{warning 'TODO: Remove all instances of bBusy and remove from VAR list in FB_StateMachine'}
FUNCTION_BLOCK FB_StateMachine IMPLEMENTS I_StateMachine
VAR_INPUT
	bActive : BOOL := TRUE;
	bErrorAck : BOOL;
	eStateSourceID : E_StateSourceID;
	
	aErrorLog : REFERENCE TO ARRAY[1..SystemConfig.MAIN_EVENT_LOG_MAX_LENGTH] OF ST_Event; //Reference to the event array initially created in MAIN
	nErrorLogIndex : REFERENCE TO UINT; //Reference to the logging index initially defined in MAIN, should be 0 at the beginning of each PLC cycle
END_VAR

VAR
	// Outer-Case State Tracking Variables
	eOuterLoopState : E_OuterLoopSM_States;
	sOuterLoopState : T_MaxString := '';
	nLastOuterLoopState : UINT := 0;	
	nOuterTempState : UINT := 0;
	sLastOuterLoopState : T_MaxString := '';
	
	// Inner-Case State Tracking Variables
	nInnerLoopState : REFERENCE TO UINT;
	sInnerLoopState : T_MaxString := '';
	nLastInnerLoopState : UINT := 0;
	nInnerTempState : UINT := 0;
	sLastInnerLoopState : T_MaxString := '';
	
	// DB Logging Stuff
	eStateMachineSourceID : E_StateSourceID;
	fbEventHandler : FB_EventHandler;
	sEventTrace	: T_MaxString := '';
	
	bBusy : BOOL;
	
//	bEnableOuterStateChanges : BOOL := SystemConfig.ENABLE_OUTER_STATE_CHANGES;
//	bEnableInnerStateChanges : BOOL := SystemConfig.ENABLE_INNER_STATE_CHANGES;
END_VAR

VAR_OUTPUT
	bError : BOOL;
	sErrorDetails : T_MaxString;			
	nErrorInTask : UINT;			
END_VAR

PROPERTY Active : BOOL
GET
Active := THIS^.bActive;
END_GET
SET
bActive := Active;
END_SET
END_PROPERTY

PROPERTY PUBLIC Busy : BOOL
GET
//Busy := isBusy();

(*
	Returns THIS^.bBusy in all cases except:
	1. We are enabled/active and transitioning to Operational - This will return FALSE until operational
	2. We are enabled/active and in Setup.
	3. We are enabled/active and in either DisablingError or DisablingInactive
*)

IF bActive THEN
	
	IF eOuterLoopState = E_OuterLoopSM_States.DisabledError THEN
		Busy := FALSE; // Not busy when active and waiting for error ack 
	ELSIF eOuterLoopState <> E_OuterLoopSM_States.Operational THEN
		Busy := TRUE; // Busy if we are active and not operational
	ELSE 
		Busy := (nInnerLoopState <> 0); // Busy In operational, if we are not idle
	END_IF
	
ELSE // NOT bActive
	
	IF eOuterLoopState = E_OuterLoopSM_States.Inactive THEN
		IF nOuterTempState =  E_OuterLoopSM_States.Inactive THEN
			Busy := FALSE; // Busy until we spend at least 1 cycle inactive
		ELSE
			Busy := TRUE; // We have spent at least 1 cycle inactive
		END_IF
	ELSIF eOuterLoopState = E_OuterLoopSM_States.DisabledError THEN
		Busy := FALSE; // Not busy while waiting for error ack
	ELSE
		Busy := TRUE; // Busy until we reach inactive state
	END_IF
	
END_IF
END_GET
END_PROPERTY

METHOD ChangeInnerState : BOOL
VAR_INPUT
	nNewState : UINT;
END_VAR
nInnerLoopState := nNewState;
END_METHOD

METHOD ChangeOuterState : BOOL
VAR_INPUT
	nNewState	: E_OuterLoopSM_States;
END_VAR
eOuterLoopState := nNewState;
END_METHOD

(*
Use the method as Case Variable ->
CASE CyclicInnerCase(TO_String(enum)) OF
1: ;
2: ;
ELSE ;
END_CASE
*)
METHOD PROTECTED CyclicInnerCase : UINT
VAR_INPUT
    sState : T_MaxString;//Name of the current state (TO_String(enum))
END_VAR
VAR_INST
    bInit : BOOL := TRUE;
END_VAR


IF (THIS^.nInnerTempState <> THIS^.nInnerLoopState) OR bInit THEN	
	// Save PreviousState
	IF bInit THEN
//		THIS^.nInnerLoopState := 0;
		THIS^.nLastInnerLoopState := THIS^.nInnerLoopState;
		THIS^.sLastInnerLoopState := sState;
		bInit := FALSE;
	ELSE
		THIS^.nLastInnerLoopState := THIS^.nInnerTempState;
		THIS^.sLastInnerLoopState := THIS^.sInnerLoopState;
		bInit := FALSE;
	END_IF
	
	// Save active State
	nInnerTempState := nInnerLoopState; 
	THIS^.sInnerLoopState := sState; //save aktive state string
	IF SystemConfig.ENABLE_INNER_STATE_CHANGES THEN
		fbEventHandler.SaveState(sLastState:=sLastInnerLoopState, sNewState:=sState, bOuter:=FALSE); //Logging after the new state has been adopted
	END_IF
END_IF


CyclicInnerCase := nInnerLoopState; //return state
END_METHOD

(*
Use the method as Case Variable ->
CASE CyclicOuterCase(TO_String(enum)) OF
1: ;
2: ;
ELSE ;
END_CASE
*)

{attribute 'monitoring':='variable'}
METHOD PRIVATE CyclicOuterCase : UINT
VAR_INPUT
    sState : T_MaxString;//Name of the current state (TO_String(enum))
END_VAR
VAR_INST
    bInit : BOOL := TRUE;
END_VAR
	
IF (THIS^.nOuterTempState <> THIS^.eOuterLoopState) OR bInit THEN

	// Save PreviousState
	IF bInit THEN
		THIS^.nLastOuterLoopState := THIS^.eOuterLoopState;
		THIS^.sLastOuterLoopState := sState;
	ELSE
		THIS^.nLastOuterLoopState := THIS^.nOuterTempState;
		THIS^.sLastOuterLoopState := THIS^.sOuterLoopState;
	END_IF
	// Save active State
	nOuterTempState := eOuterLoopState; 
	THIS^.sOuterLoopState := sState; //save aktive state string
	IF bInit THEN
		// Skips first outer state transition into setup.
		bInit := FALSE;
		
	ELSIF SystemConfig.ENABLE_OUTER_STATE_CHANGES THEN 
		fbEventHandler.SaveState(sLastState:=sLastOuterLoopState, sNewState:=sState, bOuter:=TRUE); //Logging after the new state has been adopted
	END_IF
	
END_IF


CyclicOuterCase := eOuterLoopState; //return state
END_METHOD

METHOD Disable : BOOL
// Default SUPER^.Disable method for all inheriting FBs.
// This will reset the bBusy flag and trigger an error for unimplemented Disable() methods.

fbEventHandler(eNapID:=E_Event.UNIMPLEMENTED_DISABLE_METHOD);
THIS^.bError := TRUE; // Redundant 
THIS^.bBusy := FALSE;
Disable := TRUE;
END_METHOD

PROPERTY ErrorAck : BOOL
GET
ErrorAck := bErrorAck;
END_GET
SET
bErrorAck := ErrorAck;
END_SET
END_PROPERTY

PROPERTY EventTrace : STRING
GET
EventTrace := THIS^.sEventTrace;
END_GET
END_PROPERTY

METHOD InnerLoopSM : BOOL
END_METHOD

METHOD OuterLopSM : BOOL
CASE CyclicOuterCase(sState:=TO_STRING(eOuterLoopState)) OF
	
	E_OuterLoopSM_States.Setup:
	//<<<Setup()>>>
		Setup();
		Setup_0();
		IF bActive THEN
			//<<<Reset()>>>
			Reset();
			ChangeOuterState(E_OuterLoopSM_States.Operational);
		ELSE
			ChangeOuterState(E_OuterLoopSM_States.Inactive);
		END_IF
		
	E_OuterLoopSM_States.Operational:
		IF bError THEN 
			ChangeOuterState(E_OuterLoopSM_States.DisablingError);
		ELSIF bActive THEN // No error, Active
			//<<<InnerLoopSM()>>>
			InnerLoopSM();
		ELSE // No error, not active
			ChangeOuterState(E_OuterLoopSM_States.DisablingInactive);
		END_IF

	E_OuterLoopSM_States.DisablingInactive:
		IF Disable() THEN
			ChangeOuterState(E_OuterLoopSM_States.Inactive);
		END_IF
	
	E_OuterLoopSM_States.Inactive:
		IF bActive THEN
			//<<<Reset()>>>
			//<<<ChangeInnerState(Idle)>>>
			Reset();
			ChangeInnerState(0);
			ChangeOuterState(E_OuterLoopSM_States.Operational);
		END_IF

	E_OuterLoopSM_States.DisablingError:
		IF Disable() THEN
			ChangeOuterState(E_OuterLoopSM_States.DisabledError);
		END_IF
	
	E_OuterLoopSM_States.DisabledError:
		IF bErrorAck THEN
			bError := FALSE;
			//<<<bErrorAck := FALSE>>>
			bErrorAck := FALSE;
			ChangeOuterState(E_OuterLoopSM_States.Inactive);
		END_IF
		
END_CASE
END_METHOD

METHOD Reset : BOOL
END_METHOD

METHOD PUBLIC SetInnerEnumeration : BOOL
VAR_INPUT
	nStateEnum : REFERENCE TO UINT;
END_VAR
THIS^.nInnerLoopState REF= nStateEnum; // This should pass the reference to the inner loop state enumeration variable
END_METHOD

METHOD Setup : BOOL
END_METHOD

METHOD PRIVATE Setup_0 : BOOL
VAR_INPUT
END_VAR

VAR
	nParentInnerState: STRING(INT#4);
END_VAR
fbEventHandler(aErrorLog:=aErrorLog,
					nErrorLogIndex:=nErrorLogIndex,
						eParentID:=eStateMachineSourceID,
							sParentTrace:=sEventTrace,
								sLastParentInnerState:=sLastInnerLoopState,
									sParentInnerState:=sInnerLoopState);
END_METHOD

PROPERTY StateMachineID : STRING
GET
//StateMachineID := eStateMachineSourceID;
END_GET
END_PROPERTY

END_FUNCTION_BLOCK

(* stored: Version 1.1.0.1, ProductVersion 3.1.4024.12
   POU FB_StateMachine: Id {6a5e3c2c-15ca-463d-880f-c5775b0fbcc5}, SpecialFunc None
   Folder Properties: Id {1cee6584-11c8-4121-9121-beb8e2403f7c}
   Property Active: Id {4d9542d2-fdf4-4551-be1a-1178557ec911}
   Get Get: Id {84bd4977-10df-46ae-978a-3b42c8120a31}
   Set Set: Id {10036ecc-aac9-444f-9bd3-f5f6a6991dd4}
   Property Busy: Id {c397c92b-d476-40b1-8895-b4a7aa72ae57}
   Get Get: Id {35fc2301-9d2a-4775-ae72-dcf203ff6219}
   Method ChangeInnerState: Id {61ea47ef-d8bd-428e-a0d3-2bd070ba40de}
   Method ChangeOuterState: Id {8436ae5e-f601-4561-8792-634fb7f208b5}
   Method CyclicInnerCase: Id {a3fb859c-d59d-43e7-a381-a08e5bee0551}
   Method CyclicOuterCase: Id {fab6a548-cbb6-491f-bb21-2984f49a742f}
   Method Disable: Id {ee22807d-35ad-48d7-b113-a8185df15c69}
   Property ErrorAck: Id {97eadf24-291b-4e7e-a36e-d4b50809b026}
   Get Get: Id {627898e5-a9f7-4d67-8e47-b49aa613b45a}
   Set Set: Id {085caf73-989a-413f-bac8-4428d967d718}
   Property EventTrace: Id {edbf6dc4-ea5c-4983-8228-904adbc35a0c}
   Get Get: Id {2c818f06-36fa-44d0-b6fc-59fa7b0cc03e}
   Method InnerLoopSM: Id {aa4c3d85-62e3-4797-b923-0fb9bbbd55f4}
   Method OuterLopSM: Id {32768734-abdf-415d-ac7e-7bc8b3c39e77}
   Method Reset: Id {e47b2e70-0ee6-4a26-9bab-58488c5443b6}
   Method SetInnerEnumeration: Id {dfd08693-0c3c-427d-a052-050772d7a686}
   Method Setup: Id {21afff8a-06ff-49f2-b06b-31ef6eb9d43c}
   Method Setup_0: Id {f43a19dc-99a3-439e-8bb3-d60ee2ddeb9a}
   Property StateMachineID: Id {7a34e1c6-8d0d-422d-af05-1c8585ae9791}
   Get Get: Id {64270503-62a6-4e7d-97a3-98c04c40015e} *)
